TYPE lineControlHmiCommands_TypeStruct :
STRUCT
	
	speedInc : BOOL;
	speedDec : BOOL;
	speedStop : BOOL;

END_STRUCT
END_TYPE

(* stored: Version 1.1.0.1
   DUT lineControlHmiCommands_TypeStruct: Id {c1ccb89c-be1c-40b6-9cb6-92df3ffa3874} *)
